TYPE QualityInspectionComRequest :
STRUCT
  Start : BOOL;
  Stop : BOOL;
  GoHome : BOOL;
  Halt : BOOL;
END_STRUCT
END_TYPE

(* stored: Version 1.1.0.1
   DUT QualityInspectionComRequest: Id {6a5fcf6e-58ec-4970-90e4-453053f4c30b} *)
